(* IEC 61131-3 sources: controlforge-structured-text/manual-tests/syntax, 11 files *)

(* ---- function-blocks.st ---- *)
(* Test file for FUNCTION_BLOCK syntax highlighting *)

(* Test 1: FUNCTION_BLOCK declaration with parameters *)
FUNCTION_BLOCK FB_Counter
VAR_INPUT
    increment : BOOL;
    reset : BOOL;
    maxValue : INT := 100;
END_VAR

VAR_OUTPUT
    count : INT;
    overflow : BOOL;
END_VAR

VAR
    internalState : INT;
END_VAR

// Body
IF reset THEN
    count := 0;
    overflow := FALSE;
ELSIF increment THEN
    IF count < maxValue THEN
        count := count + 1;
    ELSE
        overflow := TRUE;
    END_IF
END_IF

END_FUNCTION_BLOCK

(* Test 2: FUNCTION_BLOCK with VAR_IN_OUT *)
FUNCTION_BLOCK FB_Swap
VAR_IN_OUT
    valueA : REAL;
    valueB : REAL;
END_VAR

VAR
    temp : REAL;
END_VAR

// Swap logic
temp := valueA;
valueA := valueB;
valueB := temp;

END_FUNCTION_BLOCK

(* Test 3: Using function blocks in a PROGRAM *)
PROGRAM TestFunctionBlocks
VAR
    // Standard FB instances (should highlight TON, CTU, R_TRIG as types)
    myTimer : TON;
    myCounter : CTU;
    myEdge : R_TRIG;

    // Custom FB instances
    customCounter : FB_Counter;
    swapper : FB_Swap;

    // Test variables
    startSignal : BOOL := FALSE;
    resetSignal : BOOL := FALSE;
    result : BOOL;
    val1 : REAL := 1.5;
    val2 : REAL := 2.5;
END_VAR

// Standard FB calls with named parameters
myTimer(IN := startSignal, PT := T#5s);
myCounter(CU := myEdge.Q, R := resetSignal, PV := 10);
myEdge(CLK := startSignal);

// Custom FB calls
customCounter(increment := startSignal, reset := resetSignal, maxValue := 50);
swapper(valueA := val1, valueB := val2);

result := myTimer.Q;

END_PROGRAM

(* ---- array-of-scope.st ---- *)
(* Manual QA: OF keyword scoping in ARRAY vs CASE (#95)
   OPEN: this file in VS Code with the extension active.
   USE:  Ctrl+Shift+P -> "Developer: Inspect Editor Tokens and Scopes"

   EXPECT:
     - OF after ] in ARRAY declaration → keyword.other.array-of.st
     - OF in CASE...OF               → keyword.control.st
*)

PROGRAM ArrayOfTest
VAR
    row    : ARRAY[1..10] OF INT;       (* EXPECT: OF → keyword.other.array-of.st *)
    grid   : ARRAY[0..3, 0..3] OF REAL; (* EXPECT: OF → keyword.other.array-of.st *)
    flags  : ARRAY[
        1..100
    ] OF BOOL;                          (* EXPECT: OF → keyword.other.array-of.st *)
    x      : INT := 5;
END_VAR

CASE x OF                               (* EXPECT: OF → keyword.control.st *)
    1: x := 10;
    2: x := 20;
ELSE
    x := 0;
END_CASE

END_PROGRAM

(* ---- char-wstring-types.st ---- *)
(* Manual QA: WSTRING / CHAR / WCHAR data types (#87)
   OPEN: this file in VS Code with the extension active.
   USE:  Ctrl+Shift+P -> "Developer: Inspect Editor Tokens and Scopes"
   EXPECT: CHAR, WCHAR, WSTRING each scoped as storage.type.st
*)

PROGRAM CharTypeTest
VAR
    myChar    : CHAR    := 'A';          (* EXPECT: CHAR    → storage.type.st *)
    myWChar   : WCHAR   := "Ω";          (* EXPECT: WCHAR   → storage.type.st *)
    myString  : STRING[80] := 'hello';   (* EXPECT: STRING  → storage.type.st *)
    myWString : WSTRING[80] := "wide";   (* EXPECT: WSTRING → storage.type.st *)
END_VAR

END_PROGRAM

(* ---- hardware-addresses.st ---- *)
(* Manual QA: hardware address literals (#82)
   OPEN: this file in VS Code with the extension active.
   USE:  Ctrl+Shift+P -> "Developer: Inspect Editor Tokens and Scopes"
         hover over each %... literal and confirm the scope is
         constant.other.hardware-address.st
*)

PROGRAM HardwareAddressTest
VAR
    Input_Bit_0  AT %IX0.0  : BOOL;   (* EXPECT: %IX0.0  → constant.other.hardware-address.st *)
    Input_Bit_7  AT %IX1.7  : BOOL;   (* EXPECT: %IX1.7  → constant.other.hardware-address.st *)
    Input_Word   AT %IW2    : INT;    (* EXPECT: %IW2    → constant.other.hardware-address.st *)
    Output_Bit   AT %QX0.0  : BOOL;  (* EXPECT: %QX0.0  → constant.other.hardware-address.st *)
    Output_Word  AT %QW1    : INT;   (* EXPECT: %QW1    → constant.other.hardware-address.st *)
    Mem_DWord    AT %MD100  : DINT;  (* EXPECT: %MD100  → constant.other.hardware-address.st *)
    Mem_Byte     AT %MB5    : BYTE;  (* EXPECT: %MB5    → constant.other.hardware-address.st *)
    Mem_Long     AT %IL3    : LINT;  (* EXPECT: %IL3    → constant.other.hardware-address.st *)
    Deep_Addr    AT %IX1.2.3 : BOOL; (* EXPECT: %IX1.2.3 → constant.other.hardware-address.st *)
END_VAR

END_PROGRAM

(* ---- highlighting.st ---- *)
(* Test file for syntax highlighting verification *)
PROGRAM TestHighlighting
VAR
    // Basic types
    boolVar : BOOL := TRUE;
    intVar : INT := 123;
    realVar : REAL := 3.14;

    // Extended time types (should be highlighted now)
    timeVar : TIME := T#10s;
    ltimeVar : LTIME := LTIME#1d_2h_30m_45s;
    dateVar : DATE := D#2025-06-12;
    ldateVar : LDATE := LDATE#2025-06-12;

    // Character types (should be highlighted)
    charVar : CHAR := 'A';
    wcharVar : WCHAR := "Ω";

    // String types
    stringVar : STRING := 'Hello World';
    wstringVar : WSTRING := "Unicode String";

    // Extended integer and real types
    lwordVar : LWORD := 16#123456789ABCDEF0;
    lintVar : LINT := -9223372036854775808;
    ulintVar : ULINT := 18446744073709551615;
    lrealVar : LREAL := 2.71828182845904523536;

    // Typed numeric literals (alternative IEC 61131-3 syntax)
    typedLWord : LWORD := LWORD#16#123456789ABCDEF0;
    typedWord : WORD := WORD#16#ABCD;
    typedByte : BYTE := BYTE#16#FF;

    // Generic types
    anyVar : ANY;
    anyNumVar : ANY_NUM;
    anyRealVar : ANY_REAL;

    // Standard function block types (should be highlighted)
    myTimer : TON;
    myPulse : TP;
    myCounter : CTU;
    myEdgeDetector : R_TRIG;
    myFlipFlop : RS;

    // Loop variable
    i : INT;
END_VAR

(* Block comment test - should be highlighted as comment
   Multi-line block comments with keywords like IF THEN ELSE inside
   should not be highlighted as keywords *)

// Test control structures with highlighting
IF boolVar THEN
    intVar := intVar + 1;
    realVar := ABS(realVar);

    // Test logical operators: AND, OR, NOT, XOR
    IF boolVar AND (intVar > 50) THEN
        stringVar := 'Condition met';
    END_IF

    boolVar := (intVar > 0) OR (realVar < 0.0);
    boolVar := NOT boolVar;

    // Test MOD operator
    intVar := intVar MOD 10;

    // Test string literals with both quote styles
    stringVar := 'Single-quoted string';
    wstringVar := "Double-quoted string";

    CASE intVar OF
        1..10:
            stringVar := 'Low range';
        11..100:
            stringVar := 'Medium range';
    ELSE
        stringVar := 'High range';
    END_CASE

    FOR i := 1 TO 10 DO
        lrealVar := lrealVar * 1.1;
    END_FOR

    WHILE intVar < 100 DO
        intVar := intVar + 1;
    END_WHILE

END_IF

(* Another block comment at the end *)

END_PROGRAM

(* ---- literals.st ---- *)
(* Test file for IEC 61131-3 literal highlighting *)
PROGRAM TestLiterals
VAR
    // Time literals
    shortTime : TIME := T#10s;
    longTime : LTIME := LTIME#1d_2h_30m_45s;
    timeMs : TIME := T#500ms;
    timeUs : TIME := T#100us;
    timeNs : LTIME := LTIME#50ns;

    // Date literals
    normalDate : DATE := D#2025-06-12;
    longDate : LDATE := LDATE#2025-12-31;

    // Time of day literals
    timeOfDay : TIME_OF_DAY := TOD#14:30:15;
    longTimeOfDay : LTIME_OF_DAY := LTOD#23:59:59.999;
    timeOfDay2 : TIME_OF_DAY := TIME_OF_DAY#08:00:00;

    // Date and time literals
    dateTime : DATE_AND_TIME := DT#2025-06-12-14:30:15;
    longDateTime : LDATE_AND_TIME := LDT#2025-12-31-23:59:59.999;
    dateTime2 : DATE_AND_TIME := DATE_AND_TIME#2025-01-01-00:00:00;

    // Numeric literals (regular)
    hexValue : WORD := 16#ABCD;
    binValue : BYTE := 2#11110000;
    octValue : BYTE := 8#377;
    intValue : INT := 12345;
    realValue : REAL := 3.14159;
    expValue : REAL := 1.23E-4;

    // Typed numeric literals (IEC 61131-3 extension)
    typedByte : BYTE := BYTE#16#FF;
    typedWord : WORD := WORD#16#ABCD;
    typedDWord : DWORD := DWORD#16#12345678;
    typedLWord : LWORD := LWORD#16#123456789ABCDEF0;
    typedBinary : BYTE := BYTE#2#11110000;
    typedOctal : BYTE := BYTE#8#377;
    typedInt : INT := INT#12345;
    typedReal : REAL := REAL#3.14159;
END_VAR

// All these literals should be highlighted as complete constants,
// not split between type prefix and value
END_PROGRAM

(* ---- named-parameters.st ---- *)
(* Manual test: named parameter highlighting in FB/function calls
   Open this file in VS Code with the extension active.
   Use "Developer: Inspect Editor Tokens and Scopes" (Ctrl+Shift+P) to
   verify scope names on each token. *)

PROGRAM TestNamedParams
VAR
    MyTimer   : TON;
    MyCounter : CTU;
    StartSig  : BOOL;
    StopSig   : BOOL;
    CountOut  : INT;
    Result    : BOOL;
    Val1      : INT;
    Val2      : INT;
    i         : INT;
END_VAR

(* --- EXPECTED: named params scoped as variable.parameter.st --- *)

(* FB call with named input params: IN and PT should be variable.parameter.st *)
MyTimer(IN := StartSig, PT := T#5s);

(* FB call with named output param: Q should be variable.parameter.st, ET also *)
MyTimer(IN := StartSig, PT := T#5s, Q => Result, ET => CountOut);

(* Counter FB: CU, RESET, PV are variable.parameter.st; CV => is output *)
MyCounter(CU := StartSig, RESET := StopSig, PV := 10, CV => CountOut);

(* FB call with multiple named input params: CU, RESET, PV are variable.parameter.st *)
MyCounter(CU := Val1, RESET := StopSig, PV := Val2);

(* Multi-line call: each param name on its own line should still be variable.parameter.st *)
MyTimer(
    IN := StartSig,
    PT := T#10s
);

(* --- EXPECTED: regular assignments NOT scoped as variable.parameter.st --- *)

(* Plain assignment: i should be a plain identifier, NOT variable.parameter.st *)
i := 5;
Result := TRUE;
Val1 := Val2 + 1;

(* Variable declaration assignment: also NOT variable.parameter.st *)
(* (already shown in VAR block above) *)

END_PROGRAM

(* ---- nested-comments-test.st ---- *)
// Manual test: nested block comments (issue #84)
// Expected: all (* *) blocks highlighted as comments, including nested content

// Level 1 — single block comment (baseline)
(* This is a simple block comment *)

// Level 2 — one level of nesting; entire line highlighted as comment
(* outer comment (* inner comment *) back to outer *)

// Level 3 — two levels of nesting
(* outer (* middle (* inner *) middle *) outer *)

// Inline — nested comment alongside real code; everything inside (* *) is highlighted as comment
PROGRAM NestedCommentTest
    VAR
        x : INT; (* inline comment *)
        y : INT; (* outer (* nested *) ouDter *)
    END_VAR

    (* This comment spans
   multiple lines
   (* with a nested comment inside *)
    AND continues after *)
    x := 1;

    // Line comments unaffected
    // (* this is a line comment, not a block comment *)

END_PROGRAM

(* ---- pragmas.st ---- *)
(* Manual QA: pragma / attribute blocks (#81)
   OPEN: this file in VS Code with the extension active.
   USE:  Ctrl+Shift+P -> "Developer: Inspect Editor Tokens and Scopes"

   EXPECT for every {…} block:
     - entire block scoped as  meta.pragma.st
     - { and } scoped as       punctuation.definition.pragma.begin/end.st
     - directive keyword inside scoped as  keyword.other.pragma.st
     - string literals inside  highlighted normally (string.quoted.single etc.)
*)

{attribute 'qualified_only'}
{attribute 'hide'}
{attribute 'obsolete' := 'Use NewFB instead'}
{warning 'disable' '95'}

{region 'Motor Control Logic'}
(* code here *)
{endregion}

{IF defined(SIMULATION_MODE)}
(* simulation-only code *)
{ELSE}
(* hardware code *)
{ENDIF}

PROGRAM PragmaTest
{attribute 'no_check'}
VAR
    x : INT := 0;
END_VAR

x := x + 1;

END_PROGRAM

(* ---- test.iecst ---- *)
(* Manual test: .iecst file extension support
   This file verifies the extension activates for .iecst files.
   Expected: syntax highlighting, diagnostics, completion, and all
   LSP features work identically to .st files. *)

PROGRAM IecstExtensionTest
VAR
    counter : INT := 0;
    running : BOOL := TRUE;
    temperature : REAL := 22.5;
    message : STRING := 'Hello from .iecst';
END_VAR

(* Verify syntax highlighting works *)
IF running THEN
    counter := counter + 1;
    IF counter > 100 THEN
        running := FALSE;
    END_IF
END_IF

(* Verify completion works — type "cou" and expect "counter" *)
(* Verify diagnostics — uncomment next line for missing semicolon *)
// temperature := 50.0

(* Verify hover — hover on TON below *)
// timerInstance : TON;

CASE counter OF
    1: message := 'One';
    2: message := 'Two';
ELSE
    message := 'Other';
END_CASE

FOR counter := 1 TO 10 DO
    temperature := temperature + 0.1;
END_FOR

END_PROGRAM

(* ---- test.st ---- *)
PROGRAM ProgramName
VAR
    variable : INT := 0;
END_VAR

// Program code

END_PROGRAM
